Omron CX-Programmer project NewProject (CX-Programmer 9.61)

# PLC tujuhsegment: CP1L M

## Global symbols (name address type ; comment)
0.00 BOOL  ; TOMBOL
0.01 BOOL  ; matikan
100.00 BOOL  ; sA
100.01 BOOL  ; sB
100.02 BOOL  ; sC
100.03 BOOL  ; sD
100.04 BOOL  ; sE
100.05 BOOL  ; sF
100.06 BOOL  ; sG
10.00 BOOL  ; A
10.01 BOOL  ; B
10.02 BOOL  ; C
10.03 BOOL  ; D
10.04 BOOL  ; E
10.05 BOOL  ; F
10.06 BOOL  ; G
10.07 BOOL  ; H
10.08 BOOL  ; I
10.09 BOOL  ; J
20.00 BOOL  ; bantu1
20.01 BOOL  ; bantu2
20.02 BOOL  ; bantu3
20.03 BOOL  ; bantu4
20.04 BOOL  ; bantu5
20.05 BOOL  ; bantu6
20.06 BOOL  ; bantu7
20.07 BOOL  ; bantu8
20.08 BOOL  ; bantu9
20.09 BOOL  ; bantu10
20.10 BOOL  ; bantu11
20.11 BOOL  ; bantu12
20.12 BOOL  ; bantu13
20.13 BOOL  ; bantu14
20.14 BOOL  ; bantu15
20.15 BOOL  ; bantu16
30.00 BOOL  ; tahan
30.01 BOOL  ; tahan 2
40.00 BOOL  ; bantu17
40.01 BOOL  ; bantu18
40.02 BOOL  ; bantu19
40.03 BOOL  ; bantu20
40.04 BOOL  ; bantu21
50.00 BOOL  ; tahan
50.01 BOOL  ; tahan
50.02 BOOL  ; tahan
50.03 BOOL  ; tahan
50.04 BOOL  ; tahan
50.05 BOOL  ; tahan
50.06 BOOL  ; tahan
50.07 BOOL  ; tahan
50.08 BOOL  ; tahan
50.09 BOOL  ; tahan

## Program NewProgram1 (cyclic task 0)

### Section Section1

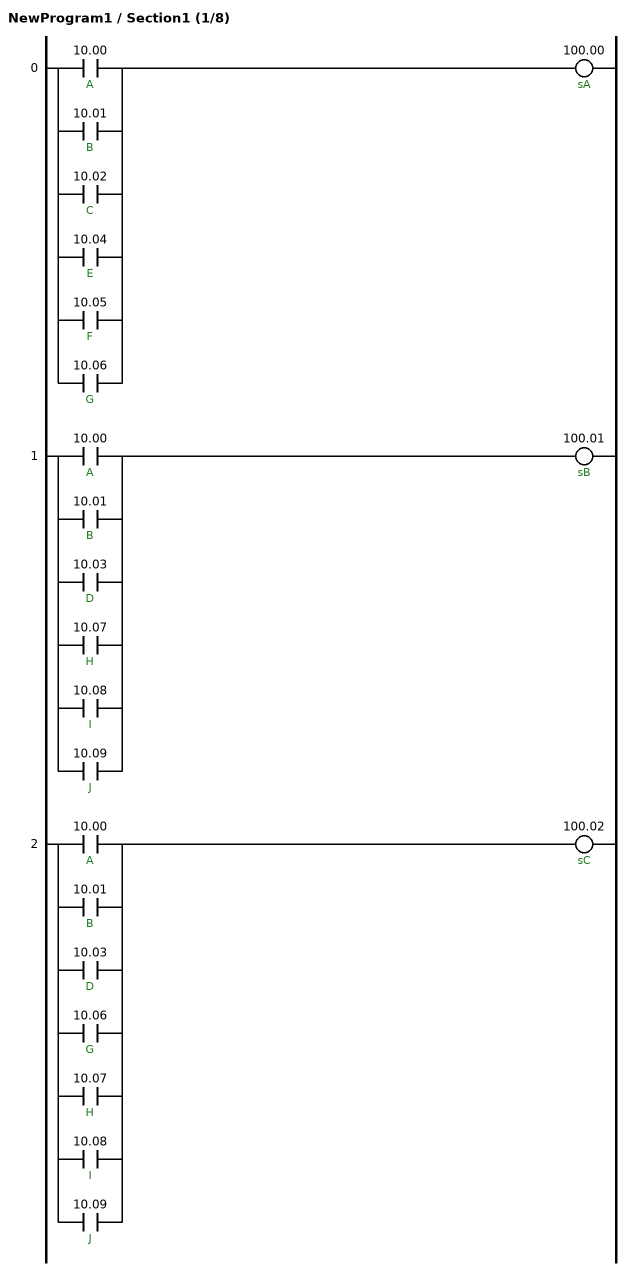
; rung 0
LD 10.00  ; A
OR 10.01  ; B
OR 10.02  ; C
OR 10.04  ; E
OR 10.05  ; F
OR 10.06  ; G
OUT 100.00  ; sA
; rung 1
LD 10.00  ; A
OR 10.01  ; B
OR 10.03  ; D
OR 10.07  ; H
OR 10.08  ; I
OR 10.09  ; J
OUT 100.01  ; sB
; rung 2
LD 10.00  ; A
OR 10.01  ; B
OR 10.03  ; D
OR 10.06  ; G
OR 10.07  ; H
OR 10.08  ; I
OR 10.09  ; J
OUT 100.02  ; sC

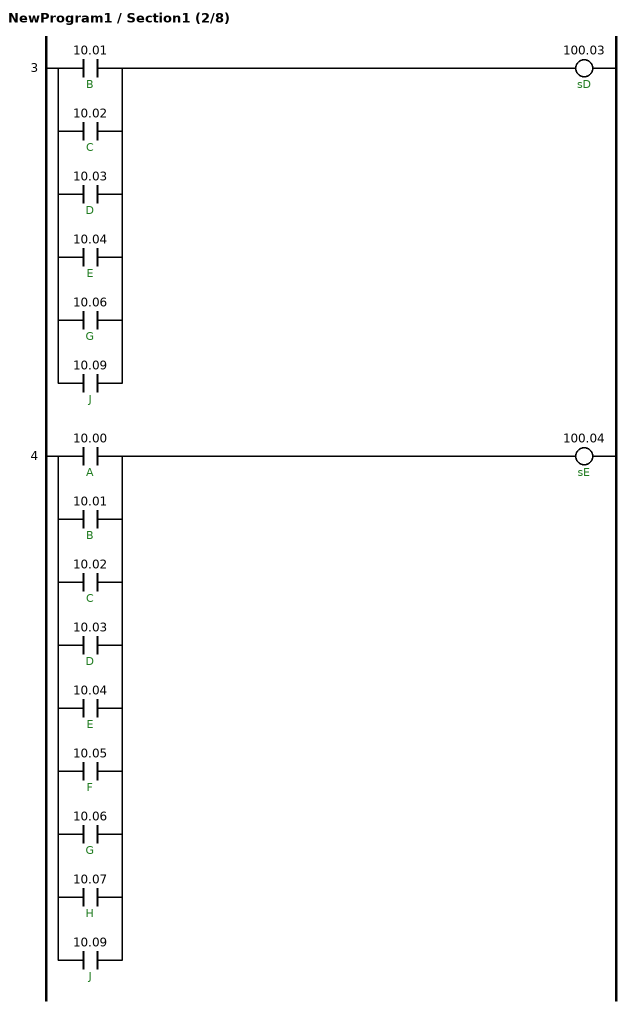
; rung 3
LD 10.01  ; B
OR 10.02  ; C
OR 10.03  ; D
OR 10.04  ; E
OR 10.06  ; G
OR 10.09  ; J
OUT 100.03  ; sD
; rung 4
LD 10.00  ; A
OR 10.01  ; B
OR 10.02  ; C
OR 10.03  ; D
OR 10.04  ; E
OR 10.05  ; F
OR 10.06  ; G
OR 10.07  ; H
OR 10.09  ; J
OUT 100.04  ; sE

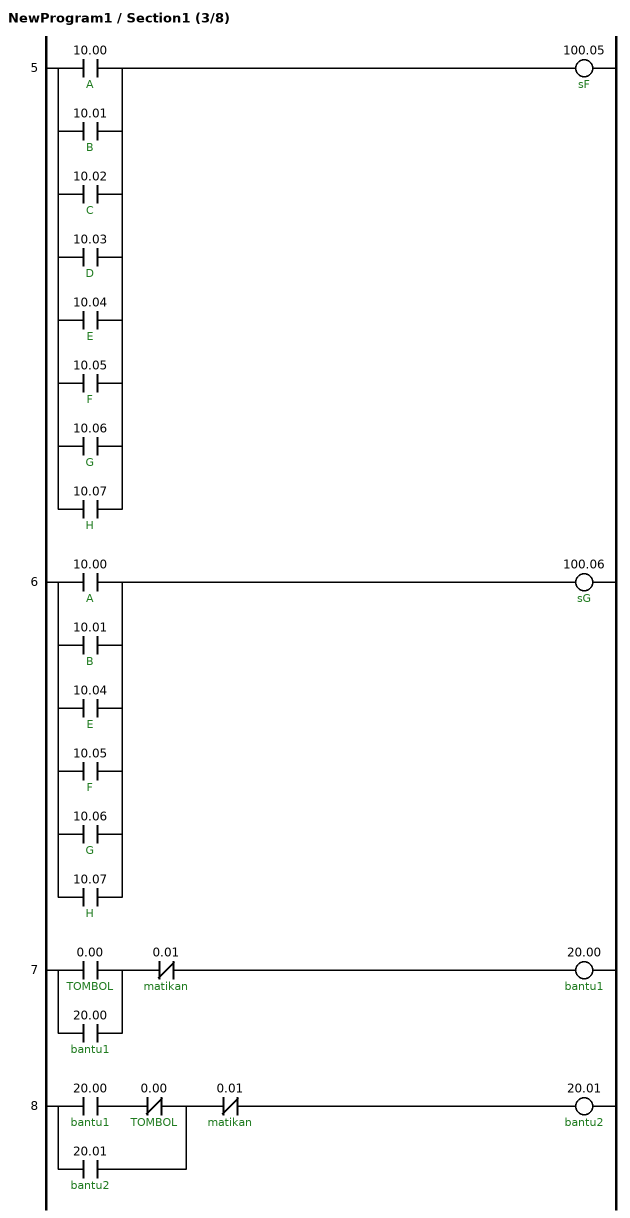
; rung 5
LD 10.00  ; A
OR 10.01  ; B
OR 10.02  ; C
OR 10.03  ; D
OR 10.04  ; E
OR 10.05  ; F
OR 10.06  ; G
OR 10.07  ; H
OUT 100.05  ; sF
; rung 6
LD 10.00  ; A
OR 10.01  ; B
OR 10.04  ; E
OR 10.05  ; F
OR 10.06  ; G
OR 10.07  ; H
OUT 100.06  ; sG
; rung 7
LD 0.00  ; TOMBOL
OR 20.00  ; bantu1
ANDNOT 0.01  ; matikan
OUT 20.00  ; bantu1
; rung 8
LD 20.00  ; bantu1
ANDNOT 0.00  ; TOMBOL
OR 20.01  ; bantu2
ANDNOT 0.01  ; matikan
OUT 20.01  ; bantu2

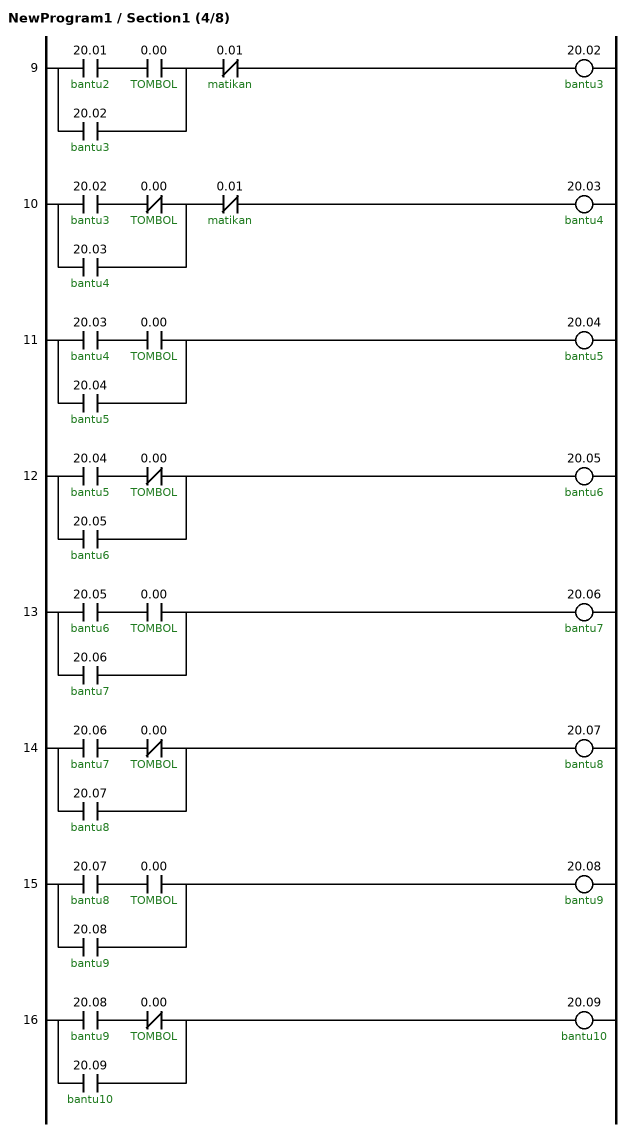
; rung 9
LD 20.01  ; bantu2
AND 0.00  ; TOMBOL
OR 20.02  ; bantu3
ANDNOT 0.01  ; matikan
OUT 20.02  ; bantu3
; rung 10
LD 20.02  ; bantu3
ANDNOT 0.00  ; TOMBOL
OR 20.03  ; bantu4
ANDNOT 0.01  ; matikan
OUT 20.03  ; bantu4
; rung 11
LD 20.03  ; bantu4
AND 0.00  ; TOMBOL
OR 20.04  ; bantu5
OUT 20.04  ; bantu5
; rung 12
LD 20.04  ; bantu5
ANDNOT 0.00  ; TOMBOL
OR 20.05  ; bantu6
OUT 20.05  ; bantu6
; rung 13
LD 20.05  ; bantu6
AND 0.00  ; TOMBOL
OR 20.06  ; bantu7
OUT 20.06  ; bantu7
; rung 14
LD 20.06  ; bantu7
ANDNOT 0.00  ; TOMBOL
OR 20.07  ; bantu8
OUT 20.07  ; bantu8
; rung 15
LD 20.07  ; bantu8
AND 0.00  ; TOMBOL
OR 20.08  ; bantu9
OUT 20.08  ; bantu9
; rung 16
LD 20.08  ; bantu9
ANDNOT 0.00  ; TOMBOL
OR 20.09  ; bantu10
OUT 20.09  ; bantu10

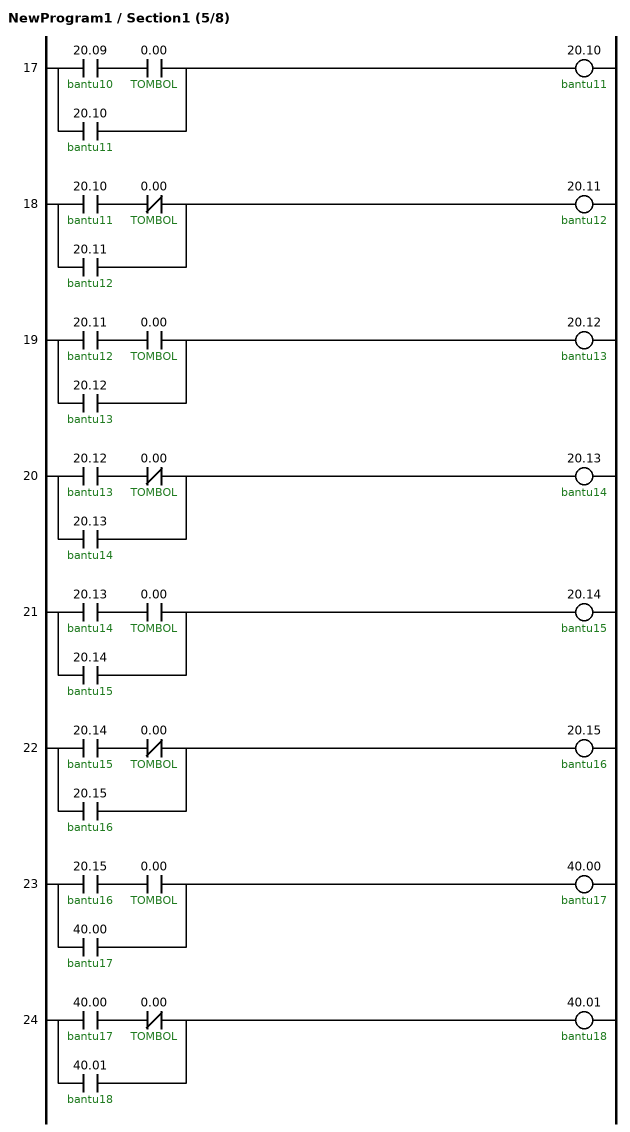
; rung 17
LD 20.09  ; bantu10
AND 0.00  ; TOMBOL
OR 20.10  ; bantu11
OUT 20.10  ; bantu11
; rung 18
LD 20.10  ; bantu11
ANDNOT 0.00  ; TOMBOL
OR 20.11  ; bantu12
OUT 20.11  ; bantu12
; rung 19
LD 20.11  ; bantu12
AND 0.00  ; TOMBOL
OR 20.12  ; bantu13
OUT 20.12  ; bantu13
; rung 20
LD 20.12  ; bantu13
ANDNOT 0.00  ; TOMBOL
OR 20.13  ; bantu14
OUT 20.13  ; bantu14
; rung 21
LD 20.13  ; bantu14
AND 0.00  ; TOMBOL
OR 20.14  ; bantu15
OUT 20.14  ; bantu15
; rung 22
LD 20.14  ; bantu15
ANDNOT 0.00  ; TOMBOL
OR 20.15  ; bantu16
OUT 20.15  ; bantu16
; rung 23
LD 20.15  ; bantu16
AND 0.00  ; TOMBOL
OR 40.00  ; bantu17
OUT 40.00  ; bantu17
; rung 24
LD 40.00  ; bantu17
ANDNOT 0.00  ; TOMBOL
OR 40.01  ; bantu18
OUT 40.01  ; bantu18

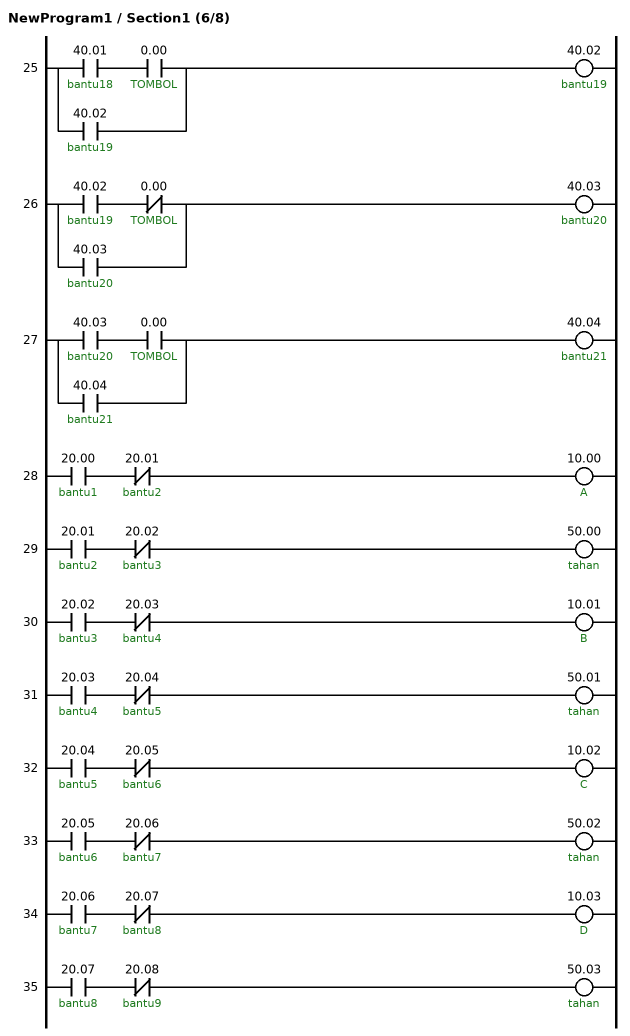
; rung 25
LD 40.01  ; bantu18
AND 0.00  ; TOMBOL
OR 40.02  ; bantu19
OUT 40.02  ; bantu19
; rung 26
LD 40.02  ; bantu19
ANDNOT 0.00  ; TOMBOL
OR 40.03  ; bantu20
OUT 40.03  ; bantu20
; rung 27
LD 40.03  ; bantu20
AND 0.00  ; TOMBOL
OR 40.04  ; bantu21
OUT 40.04  ; bantu21
; rung 28
LD 20.00  ; bantu1
ANDNOT 20.01  ; bantu2
OUT 10.00  ; A
; rung 29
LD 20.01  ; bantu2
ANDNOT 20.02  ; bantu3
OUT 50.00  ; tahan
; rung 30
LD 20.02  ; bantu3
ANDNOT 20.03  ; bantu4
OUT 10.01  ; B
; rung 31
LD 20.03  ; bantu4
ANDNOT 20.04  ; bantu5
OUT 50.01  ; tahan
; rung 32
LD 20.04  ; bantu5
ANDNOT 20.05  ; bantu6
OUT 10.02  ; C
; rung 33
LD 20.05  ; bantu6
ANDNOT 20.06  ; bantu7
OUT 50.02  ; tahan
; rung 34
LD 20.06  ; bantu7
ANDNOT 20.07  ; bantu8
OUT 10.03  ; D
; rung 35
LD 20.07  ; bantu8
ANDNOT 20.08  ; bantu9
OUT 50.03  ; tahan

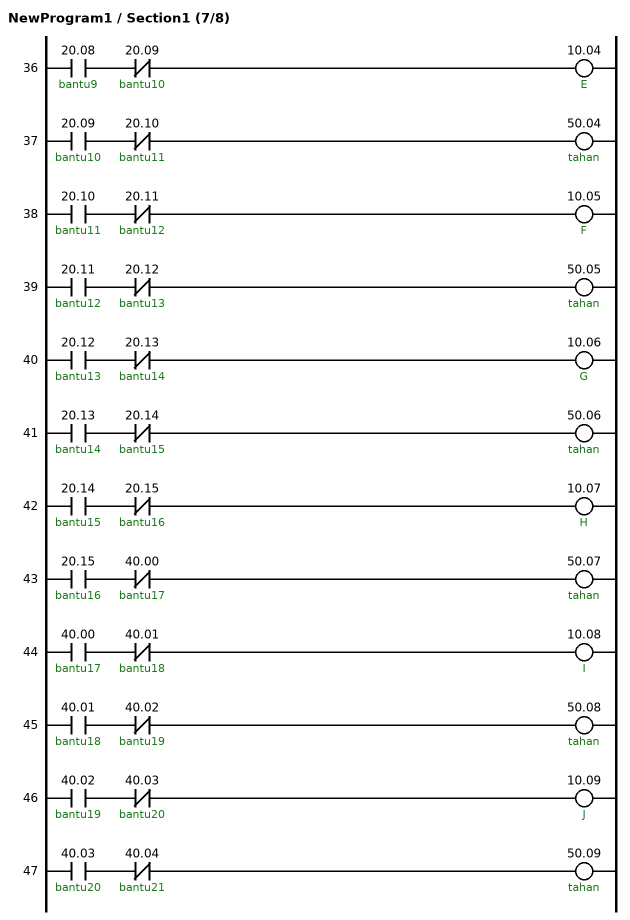
; rung 36
LD 20.08  ; bantu9
ANDNOT 20.09  ; bantu10
OUT 10.04  ; E
; rung 37
LD 20.09  ; bantu10
ANDNOT 20.10  ; bantu11
OUT 50.04  ; tahan
; rung 38
LD 20.10  ; bantu11
ANDNOT 20.11  ; bantu12
OUT 10.05  ; F
; rung 39
LD 20.11  ; bantu12
ANDNOT 20.12  ; bantu13
OUT 50.05  ; tahan
; rung 40
LD 20.12  ; bantu13
ANDNOT 20.13  ; bantu14
OUT 10.06  ; G
; rung 41
LD 20.13  ; bantu14
ANDNOT 20.14  ; bantu15
OUT 50.06  ; tahan
; rung 42
LD 20.14  ; bantu15
ANDNOT 20.15  ; bantu16
OUT 10.07  ; H
; rung 43
LD 20.15  ; bantu16
ANDNOT 40.00  ; bantu17
OUT 50.07  ; tahan
; rung 44
LD 40.00  ; bantu17
ANDNOT 40.01  ; bantu18
OUT 10.08  ; I
; rung 45
LD 40.01  ; bantu18
ANDNOT 40.02  ; bantu19
OUT 50.08  ; tahan
; rung 46
LD 40.02  ; bantu19
ANDNOT 40.03  ; bantu20
OUT 10.09  ; J
; rung 47
LD 40.03  ; bantu20
ANDNOT 40.04  ; bantu21
OUT 50.09  ; tahan

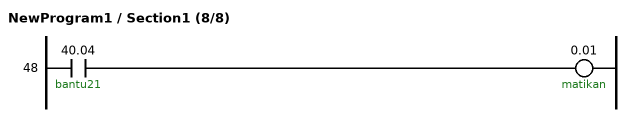
; rung 48
LD 40.04  ; bantu21
OUT 0.01  ; matikan

### Section END
; rung 0
END(001)